// SIMATIC STEP 7 (V5.x) project Project
// CPU: CPU 315-2 DP
// CPU: CPU 315-2 DP
// station: Hardware
// station: SIMATIC 300(1)
// station: P_ADR_BUS
// station: Hardware
// station: SIMATIC 300(2)
// station: P_ADR_BUS
// station: _S7H_BUSSYSTEM_CT
// station: _S7H_BUSSYSTEM_CT
// program: S7 Program(1)
// program: S7 Program(1)

SYMBOL_TABLE
"A_Sensors"	DB 2	DB 2
"DI"	DB 3	DB 3
"SensorsSettings"	DB 4	DB 4
"Valves"	DB 5	DB 5
"BD_Coils"	DB 6	DB 6
"KB1_1_Coils"	DB 7	DB 7
"KB1_2_Coils"	DB 8	DB 8
"KB2_Coils"	DB 9	DB 9
"PO1_1_Coils"	DB 10	DB 10
"PO1_2_Coils"	DB 11	DB 11
"GA1_1_Coils"	DB 12	DB 12
"GA1_2_Coils"	DB 13	DB 13
"GA2_1_Coils"	DB 14	DB 14
"GA2_2_Coils"	DB 15	DB 15
"BD_AI_1"	DB 16	DB 16
"KB1_1_AI_1"	DB 17	DB 17
"KB1_1_AI_2"	DB 18	DB 18
"KB1_1_AI_3"	DB 19	DB 19
"KB1_2_AI_1"	DB 20	DB 20
"KB1_2_AI_2"	DB 21	DB 21
"KB1_2_AI_3"	DB 22	DB 22
"KB2_AI_1"	DB 23	DB 23
"KB2_AI_2"	DB 24	DB 24
"KB2_AI_3"	DB 25	DB 25
"KB2_AI_4"	DB 26	DB 26
"PO1_1_AI"	DB 27	DB 27
"PO1_2_AI"	DB 28	DB 28
"GA1_1_AI_1"	DB 29	DB 29
"GA1_1_AI_2"	DB 30	DB 30
"GA1_2_AI_1"	DB 31	DB 31
"GA1_2_AI_2"	DB 32	DB 32
"GA2_1_AI_1"	DB 33	DB 33
"GA2_1_AI_2"	DB 34	DB 34
"KD1_1_AI"	DB 35	DB 35
"GA2_2_AI_1"	DB 36	DB 36
"GA2_2_AI_2"	DB 37	DB 37
"KD1_1_AI_2"	DB 38	DB 38
"KD1_1_AI_3"	DB 39	DB 39
"KD1_1_AI_4"	DB 40	DB 40
"KD1_1_AI_5"	DB 41	DB 41
"KD1_1_Coils"	DB 42	DB 42
"BD1_ARR_AI"	DB 43	DB 43
"BD_AI_2"	DB 44	DB 44
"BD_AI_3"	DB 45	DB 45
"BD_DO_1"	DB 46	DB 46
"BD_DO_2"	DB 47	DB 47
"GA1_1_DO"	DB 48	DB 48
"GA1_2_DO"	DB 49	DB 49
"GA2_1_DO"	DB 50	DB 50
"GA2_2_DO"	DB 51	DB 51
"BD_REAL"	DB 52	DB 52
"KB1_1_REAL"	DB 53	DB 53
"KB1_2_REAL"	DB 54	DB 54
"KB2_REAL"	DB 55	DB 55
"PO1_1_REAL"	DB 56	DB 56
"PO1_2_REAL"	DB 57	DB 57
"GA1_1_REAL"	DB 58	DB 58
"GA1_2_REAL"	DB 59	DB 59
"GA2_1_REAL"	DB 60	DB 60
"GA2_2_REAL"	DB 61	DB 61
"KD_REAL"	DB 62	DB 62
"ModbusVars"	DB 63	DB 63
"BD_Outputs_1"	DB 64	DB 64
"BD_Outputs_2"	DB 65	DB 65
"PO1_1_Outputs"	DB 66	DB 66
"PO1_2_Outputs"	DB 67	DB 67
"GA1_1_Outputs"	DB 68	DB 68
"GA1_2_Outputs"	DB 69	DB 69
"GA2_1_Outputs"	DB 97	DB 97
"GA2_2_Outputs"	DB 98	DB 98
"BD_OutputBytes_1"	DB 99	DB 99
"BD_OutputBytes_2"	DB 111	DB 111
"PO1_1_OutBytes"	DB 112	DB 112
"PO1_2_OutBytes"	DB 113	DB 113
"GA1_1_OutBytes"	DB 114	DB 114
"GA1_2_OutBytes"	DB 115	DB 115
"GA2_1_OutBytes"	DB 116	DB 116
"GA2_2_OutBytes"	DB 117	DB 117
"StartStop"	DB 118	DB 118
"StartStopBytes"	DB 119	DB 119
"KB2_AI_Bearer"	DB 128	DB 128
"KB2_AI_Vibration"	DB 129	DB 129
"ModbusAddresses"	DB 130	DB 130
"PO2_AI"	DB 131	DB 131
"PO2_Reals"	DB 132	DB 132
"PO2_AI2"	DB 133	DB 133
"DI_Bytes"	DB 134	DB 134
"PCV10_PID_Vars"	DB 135	DB 135
"PCV21_PID_Vars"	DB 136	DB 136
"PCV22_PID_Vars"	DB 137	DB 137
"PCV25_PID_Vars"	DB 138	DB 138
"ValvesVars"	DB 139	DB 139
"SensorsAlarmSettings"	DB 140	DB 140
"BD_MaxMin"	DB 141	DB 141
"GA1_1_MinMax"	DB 142	DB 142
"GA1_2_MinMax"	DB 143	DB 143
"GA2_1_MinMax"	DB 144	DB 144
"GA2_2_MinMax"	DB 145	DB 145
"KB1_1_MinMax"	DB 146	DB 146
"KB1_2_MinMax"	DB 147	DB 147
"KD2_ManMax"	DB 148	DB 148
"PO1_1_MaxMin"	DB 149	DB 149
"PO1_2_MinMax"	DB 150	DB 150
"ProcessSettings"	DB 151	DB 151
"ProcessVars"	DB 152	DB 152
"PrepareStartStop"	DB 153	DB 153
"PO2_Coils"	DB 154	DB 154
"PO2_MinMax"	DB 155	DB 155
"SensorsErr"	DB 156	DB 156
"DB_DO"	DB 157	DB 157
"SensorsWarningSettings"	DB 158	DB 158
"VentVars"	DB 159	DB 159
"BD_Warnings"	DB 160	DB 160
"GA1_1_Warnings"	DB 161	DB 161
"GA1_2_Warnings"	DB 162	DB 162
"GA2_2_Warnings"	DB 163	DB 163
"GA2_1_Warnings"	DB 164	DB 164
"KB1_1_Warnings"	DB 165	DB 165
"KB1_2_Warnings"	DB 166	DB 166
"KD2_Warnings"	DB 167	DB 167
"KB2_MinMax"	DB 168	DB 168
"KB2_Warnings"	DB 169	DB 169
"PO1_1_Warnings"	DB 170	DB 170
"PO1_2_Warnings"	DB 171	DB 171
"PO2_Warnings"	DB 172	DB 172
"ModbusConnestions"	DB 173	DB 173
"KB2_Outputs"	DB 174	DB 174
"KB2_OutputBytes"	DB 175	DB 175
"KB2_CalcRealBytes"	DB 176	DB 176
"KB1_1_OutBytes"	DB 177	DB 177
"KB1_2_OutBytes"	DB 178	DB 178
"KB1_1_Outputs"	DB 179	DB 179
"KB1_2_Outputs"	DB 180	DB 180
"PO2_ArrCoils"	DB 181	DB 181
"KB2_ArrCoils"	DB 182	DB 182
"GA2_1_ArrCoils"	DB 183	DB 183
"GA2_2_ArrCoils"	DB 184	DB 184
"GA1_1_ArrCoils"	DB 185	DB 185
"GA1_2_ArrCoils"	DB 186	DB 186
"KB1_1_ArrCoils"	DB 187	DB 187
"KB1_2_ArrCoils"	DB 188	DB 188
"KD1_1_ArrCoils"	DB 189	DB 189
"PO1_1_ArrCoils"	DB 190	DB 190
"PO1_2_ArrCoils"	DB 191	DB 191
"BD_ArrCoils"	DB 192	DB 192
"AlmLocks"	DB 193	DB 193
"KB2_Resistance_Block"	DB 194	DB 194
"KB2_Resistance_Warn"	DB 195	DB 195
"GA2_2_AI_3"	DB 196	DB 196
"BlockVars"	DB 197	DB 197
"ValvesAutoManualStatus"	DB 198	DB 198
"GLV"	DB 301	DB 301
"ZB1"	DB 777	FB 38
"ZB2"	DB 778	FB 38
"ZB3"	DB 779	FB 38
"ZB4"	DB 780	FB 38
"ValvesPrgDB"	DB 781	FB 39
"KB2_AI_I_Motor"	DB 11120	DB 11120
"KB2_MotorMaxMin"	DB 11122	DB 11122
"KB2_MotorWarning"	DB 11123	DB 11123
"KB2_Motor"	DB 11199	DB 11199
"BD_GetReals"	FB 1	FB 1
"KB1_1_GetReals"	FB 2	FB 2
"KB1_2_GetReals"	FB 3	FB 3
"KB2_GetReals"	FB 4	FB 4
"PO1_1_GetReals"	FB 5	FB 5
"PO1_2_GetReals"	FB 6	FB 6
"P_RCV_RK"	FB 7	FB 7	// Receive Data / Provide Data
"P_SND_RK"	FB 8	FB 8	// Send Data / Fetch Data
"GA1_1_GetReal"	FB 9	FB 9
"MBMAREQ"	FB 10	FB 10	// MBMAREQ MODBUS MASTER REQUEST FUNCTION BLOCK
"GA1_2_GetReals"	FB 11	FB 11
"GA2_1_GetReals"	FB 12	FB 12
"GA2_2_GetReals"	FB 13	FB 13
"KD_GetReals"	FB 14	FB 14
"ModbusReal"	FB 15	FB 15
"ModbusCoils"	FB 16	FB 16
"ModbusOutputs"	FB 17	FB 17
"BD_GetOutputs"	FB 18	FB 18
"PO1_1_GetOutputs"	FB 19	FB 19
"PO1_2_GetOutputs"	FB 20	FB 20
"GA1_1_GetOutputs"	FB 21	FB 21
"GA1_2_GetOutputs"	FB 22	FB 22
"GA2_1_GetOutputs"	FB 23	FB 23
"GA2_2_GetOutputs"	FB 24	FB 24
"ModbusStartStop"	FB 25	FB 25
"GetStartStopBytes"	FB 26	FB 26
"GetAll"	FB 27	FB 27
"ModbusAll"	FB 28	FB 28
"InToVars"	FB 29	FB 29
"InToVarsST"	FB 30	FB 30
"PO2_GetReals"	FB 31	FB 31
"DI_ToVars"	FB 32	FB 32
"Valve_PID"	FB 33	FB 33
"fbPID"	FB 34	FB 34
"MBMA341"	FB 35	FB 35	// MBMA341 MODBUS MASTER COMMUNICATION FUNCTION BLOCK
"DERIVATIVE"	FB 36	FB 36
"INTEGRAL"	FB 37	FB 37
"DO_Valve"	FB 38	FB 38
"ValvesPrg"	FB 39	FB 39
"fbProcess_1"	FB 40	FB 40
"CONT_C"	FB 41	FB 41	// Continuous Control
"CONT_S"	FB 42	FB 42	// Step Control
"fbImpulsValve"	FB 43	FB 43
"fbImpulsValveSCL"	FB 44	FB 44
"prProcess"	FB 45	FB 45
"fbPO"	FB 46	FB 46
"fbKB"	FB 47	FB 47
"fbKZA"	FB 48	FB 48
"prDevices"	FB 49	FB 49
"GetCoils"	FB 50	FB 50
"Trash"	FB 51	FB 51
"VentBlock"	FB 52	FB 52
"KB2_GetOuts"	FB 53	FB 53
"fbStartStopProc"	FB 54	FB 54
"fbTON_New"	FB 55	FB 55
"fbStopDevices"	FB 56	FB 56
"fbN_O2_Block"	FB 57	FB 57
"TCONT_CP"	FB 58	FB 58	// temperature PID controller with pulse generator and self-tuning
"fbN_O2_Block_1"	FB 59	FB 59
"fbN_O2_Block_2"	FB 60	FB 60
"SET_SW_S"	FB 61	FB 61	// Set summer/winter time with status
"SWR_ZYK"	FB 101	FB 101	// Cyclic function block for Software Redundance
"SWR_SFCCOM"	FB 103	FB 103	// Communication function block for Software Redundance
"SWR_AG_COM"	FB 104	FB 104	// Communication function block for Software Redundance
"LinTrafo"	FC 1	FC 1
"fnWordPack"	FC 2	FC 2
"fnBytesToReal"	FC 3	FC 3
"fnBytesToRealOneComma"	FC 4	FC 4
"fnBytesToRealPressure"	FC 5	FC 5
"fnBytesToRealTwoComas"	FC 6	FC 6
"StartStopByte"	FC 7	FC 7
"LinTrafoInt"	FC 8	FC 8
"ByteToByte"	FC 9	FC 9
"fnRepeater"	FC 10	FC 10
"fnModbusCheckConnecrions"	FC 11	FC 11
"fnMicron"	FC 12	FC 12
"LinTrafoFlow"	FC 13	FC 13
"fnMaskByte"	FC 14	FC 14
"fnWordPackTwoComas"	FC 15	FC 15
"fnAverage"	FC 16	FC 16
"fnCbarPressure"	FC 17	FC 17
"SWR_START"	FC 100	FC 100	// Initialisation function for Software Redundance
"SWR_DIAG"	FC 102	FC 102	// Diagnostic function for Software Redundance
"_DI_XL1_QL3"	I 0.0	BOOL
"_DI_XL2_QL3"	I 0.1	BOOL
"_DI_Q3_Bad"	I 0.2	BOOL
"_DI_AB1_Working"	I 0.3	BOOL
"_DI_Kb_1_1_Working"	I 0.4	BOOL
"_DI_Kb_1_1_Alm"	I 0.5	BOOL
"_DI_Kb_1_2_Working"	I 0.6	BOOL
"_DI_Kb_1_2_Alm"	I 0.7	BOOL
"_DI_Kb_2_Working"	I 1.0	BOOL
"_DI_Kb_2_Alm"	I 1.1	BOOL
"_DI_Kd_1_Working"	I 1.2	BOOL
"_DI_Kd_1_Alm"	I 1.3	BOOL
"_DI_ZB_1_Opn"	I 1.4	BOOL
"_DI_ZB_1_Cls"	I 1.5	BOOL
"_DI_ZB_1_Local"	I 1.6	BOOL
"_DI_ZB_1_Alm"	I 1.7	BOOL
"_DI_ZB_2_Opn"	I 2.0	BOOL
"_DI_ZB_2_Cls"	I 2.1	BOOL
"_DI_ZB_2_Local"	I 2.2	BOOL
"_DI_ZB_2_Alm"	I 2.3	BOOL
"_DI_ZB_3_Opn"	I 2.4	BOOL
"_DI_ZB_3_Cls"	I 2.5	BOOL
"_DI_ZB_3_Local"	I 2.6	BOOL
"_DI_ZB_3_Alm"	I 2.7	BOOL
"_DI_EUV_001_Opn"	I 3.0	BOOL
"_DI_EUV_001_Cls"	I 3.1	BOOL
"_DI_EUV_001_Local"	I 3.2	BOOL
"_DI_EUV_001_Alm"	I 3.3	BOOL
"_DI_EUV_002_Opn"	I 3.4	BOOL
"_DI_EUV_002_Cls"	I 3.5	BOOL
"_DI_EUV_002_Local"	I 3.6	BOOL
"_DI_EUV_002_Alm"	I 3.7	BOOL
"_DI_EUV_003_Opn"	I 4.0	BOOL
"_DI_EUV_003_Cls"	I 4.1	BOOL
"_DI_EUV_003_Local"	I 4.2	BOOL
"_DI_EUV_003_Alm"	I 4.3	BOOL
"QSA_19_1_1"	I 4.4	BOOL
"QSA_23_1_1"	I 4.5	BOOL
"QSA_19_1_2"	I 4.6	BOOL
"QSA_23_1_2"	I 4.7	BOOL
"QSA_19_1_3"	I 5.0	BOOL
"QSA_23_1_3"	I 5.1	BOOL
"QSA_19_1_4"	I 5.2	BOOL
"QSA_23_1_4"	I 5.3	BOOL
"QSA_19_1_5"	I 5.4	BOOL
"QSA_23_1_5"	I 5.5	BOOL
"Q3_BAD"	I 5.6	BOOL
"AB_1_Alm"	I 5.7	BOOL
"AB_2_Working"	I 6.0	BOOL
"AB_2_Alm"	I 6.1	BOOL
"AB_3_Working"	I 6.2	BOOL
"AB_3_Alm"	I 6.3	BOOL
"AB_4_Working"	I 6.4	BOOL
"AB_4_Alm"	I 6.5	BOOL
"P2_Alm"	I 6.6	BOOL
"P2_Working"	I 6.7	BOOL
"P3_Alm"	I 7.0	BOOL
"P3_Working"	I 7.1	BOOL
"IBP_1_Working"	I 7.2	BOOL
"IBP_1_Alm"	I 7.3	BOOL
"IBP_1_Bypas"	I 7.4	BOOL
"IBP_2_Working"	I 7.5	BOOL
"IBP_2_Alm"	I 7.6	BOOL
"IBP_2_Bypas"	I 7.7	BOOL
"_DI_ZB_4_Opn"	I 8.0	BOOL
"_DI_ZB_4_Cls"	I 8.1	BOOL
"_DI_ZB_4_Local"	I 8.2	BOOL
"_DI_ZB_4_Alm"	I 8.3	BOOL
"XL1_Q4"	I 8.4	BOOL
"XL2_Q4"	I 8.5	BOOL
"Q4_BAD"	I 8.6	BOOL
"_KB_1_1_1PIR7"	IW 256	WORD
"_KB_1_2_2PIR7"	IW 258	WORD
"_1PIR6"	IW 260	WORD
"_KZA_1_2_2PIR6"	IW 262	WORD
"_KB_2_PIR8"	IW 264	WORD
"_1PIR20"	IW 266	WORD
"_2PIR20"	IW 268	WORD
"_TIR10"	IW 270	WORD
"_FIR10"	IW 272	WORD
"_PIR5"	IW 274	WORD
"_FIR5"	IW 276	WORD
"_PIRC21"	IW 278	WORD
"_1PIR27"	IW 280	WORD
"_QIRAH3"	IW 282	WORD
"_2PIR27"	IW 284	WORD
"_PIR4"	IW 286	WORD
"_FIR_4"	IW 288	WORD
"_PIRC22"	IW 290	WORD
"_PIRC23"	IW 292	WORD
"_PIRC24"	IW 294	WORD
"_PIRC25"	IW 296	WORD
"_FIR_25"	IW 298	WORD
"_1PIRC26"	IW 300	WORD
"_2PIRC26"	IW 302	WORD
"_C10"	IW 304	WORD
"_TIR5"	IW 306	WORD
"_TIR4"	IW 308	WORD
"_TIR25"	IW 310	WORD
"_AIR1"	IW 312	WORD
"_QIRAH4Q4"	IW 314	WORD
"CYC_INT5"	OB 35	OB 35	// Cyclic Interrupt 5
"CYCL_FLT"	OB 80	OB 80	// Cycle Time Fault
"I/O_FLT1"	OB 82	OB 82	// I/O Point Fault 1
"OBNL_FLT"	OB 85	OB 85	// OB Not Loaded Fault
"RACK_FLT"	OB 86	OB 86	// Loss of Rack Fault
"COMM_FLT"	OB 87	OB 87	// Communication Fault
"COMPLETE RESTART"	OB 100	OB 100	// Complete Restart
"PROG_ERR"	OB 121	OB 121	// Programming Error
"MOD_ERR"	OB 122	OB 122	// Module Access Error
"_DO_HS1Q1_Acknow"	Q 0.0	BOOL
"_DO_HS1Q1_Check"	Q 0.1	BOOL
"_DO_KB_1_1_Stop"	Q 0.2	BOOL
"_DO_KB_1_1_Start"	Q 0.3	BOOL
"_DO_KB_1_2_Stop"	Q 0.4	BOOL
"_DO_KB_1_2_Start"	Q 0.5	BOOL
"_DO_KB_2_Stop"	Q 0.6	BOOL
"_DO_KB_2_Start"	Q 0.7	BOOL
"_DO_KD_1_Start"	Q 1.0	BOOL
"_DO_KD_1_Stop"	Q 1.1	BOOL
"_DO_ZB_1_CmdOpn"	Q 1.2	BOOL
"_DO_ZB_1_CmdCls"	Q 1.3	BOOL
"_DO_ZB_1_CmdStop"	Q 1.4	BOOL
"_DO_ZB_2_CmdOpn"	Q 1.5	BOOL
"_DO_ZB_2_CmdCls"	Q 1.6	BOOL
"_DO_ZB_2_CmdStop"	Q 1.7	BOOL
"_DO_ZB_3_CmdOpn"	Q 2.0	BOOL
"_DO_ZB_3_CmdCls"	Q 2.1	BOOL
"_DO_ZB_3_CmdStop"	Q 2.2	BOOL
"_DO_AlnVent"	Q 2.3	BOOL
"_DO_ZB_4_CmdOpn"	Q 2.4	BOOL
"_DO_ZB_4_CmdCls"	Q 2.5	BOOL
"_DO_ZB_4_CmdStop"	Q 2.6	BOOL
"_AO_N_Set_PCV10"	QW 256	WORD
"_AO_N_Set_PCV21"	QW 258	WORD
"_AO_Air_Set_PCV22"	QW 260	WORD
"_AO_Air_Set_PCV25"	QW 262	WORD
"TP"	SFB 3	SFB 3	// Generate a Pulse
"RDREC"	SFB 52	SFB 52	// Read a Process Data Record
"WRREC"	SFB 53	SFB 53	// Write a Process Data Record
"READ_CLK"	SFC 1	SFC 1	// Read System Clock
"GADR_LGC"	SFC 5	SFC 5	// Query Logical Address of a Channel
"RD_SINFO"	SFC 6	SFC 6	// Read OB Start Information
"DP_PRAL"	SFC 7	SFC 7	// Triggering a Hardware Interrupt on the DP Master
"EN_MSG"	SFC 9	SFC 9	// Enable Block-Related, Symbol-Related and Group Status Messages
"DIS_MSG"	SFC 10	SFC 10	// Disable Block-Related, Symbol-Related and Group Status Messages
"DPSYC_FR"	SFC 11	SFC 11	// Sending Control Commands to Groups of DP Slaves
"DPNRM_DG"	SFC 13	SFC 13	// Read Diagnostic Data of a DP Slave
"DPRD_DAT"	SFC 14	SFC 14	// Read Consistent Data of a Standard DP Slave
"DPWR_DAT"	SFC 15	SFC 15	// Write Consistent Data to a Standard DP Slave
"ALARM_SQ"	SFC 17	SFC 17	// Generate Block-Related Messages with Acknowledgment
"ALARM_S"	SFC 18	SFC 18	// Generate Permanently Acknowledged Block-Related Messages
"ALARM_SC"	SFC 19	SFC 19	// Query the Acknowledgment Status of the last ALARM_SQ Entering State Message
"BLKMOV"	SFC 20	SFC 20	// Copy Variables
"FILL"	SFC 21	SFC 21	// Initialize a Memory Area
"CREAT_DB"	SFC 22	SFC 22	// Create Data Block
"DEL_DB"	SFC 23	SFC 23	// Delete Data Block
"TEST_DB"	SFC 24	SFC 24	// Test Data Block
"COMPRESS"	SFC 25	SFC 25	// Compress the User Memory
"UPDAT_PI"	SFC 26	SFC 26	// Update Process Image Input
"UPDAT_PO"	SFC 27	SFC 27	// Update Outputs on I/O Module
"SET_TINT"	SFC 28	SFC 28	// Set Time-of-Day Interrupt
"CAN_TINT"	SFC 29	SFC 29	// Cancel Time-of-Day Interrupt
"ACT_TINT"	SFC 30	SFC 30	// Activate Time-of-Day Interrupt
"QRY_TINT"	SFC 31	SFC 31	// Query Time-of-Day Interrupt
"SRT_DINT"	SFC 32	SFC 32	// Start Time-Delay Interrupt
"CAN_DINT"	SFC 33	SFC 33	// Cancel Time-Delay Interrupt
"QRY_DINT"	SFC 34	SFC 34	// Query Time-Delay Interrupt
"MP_ALM"	SFC 35	SFC 35	// Trigger Multicomputing Interrupt
"MSK_FLT"	SFC 36	SFC 36	// Mask Synchronous Errors
"DMSK_FLT"	SFC 37	SFC 37	// Unmask Synchronous Errors
"READ_ERR"	SFC 38	SFC 38	// Read Error Registers
"DIS_IRT"	SFC 39	SFC 39	// Disable New Interrupts and Asynchronous Errors
"EN_IRT"	SFC 40	SFC 40	// Enable New Interrupts and Asynchronous Errors
"DIS_AIRT"	SFC 41	SFC 41	// Delay the Higher Priority Interrupts and Asynchronous Errors
"EN_AIRT"	SFC 42	SFC 42	// Enable Higher Priority Interrupts and Asynchronous Errors
"RE_TRIGR"	SFC 43	SFC 43	// Retrigger Cycle Time Monitoring
"REPL_VAL"	SFC 44	SFC 44	// Transfer Substitute Value to Accumulator 1
"STP"	SFC 46	SFC 46	// Change the CPU to STOP
"WAIT"	SFC 47	SFC 47	// Delay Execution of the User Program
"SNC_RTCB"	SFC 48	SFC 48	// Synchronize Slave Clocks
"LGC_GADR"	SFC 49	SFC 49	// Query the Module Slot Belonging to a Logical Address
"RD_LGADR"	SFC 50	SFC 50	// Read All Logical Addresses of a Module
"RDSYSST"	SFC 51	SFC 51	// Read a System Status List or Partial List
"WR_USMSG"	SFC 52	SFC 52	// Write a User-Defined Diagnostic Event to the Diagnostic Buffer
"RD_DPARM"	SFC 54	SFC 54	// Reading Predefined Parameters
"WR_PARM"	SFC 55	SFC 55	// Write Dynamic Parameters
"WR_DPARM"	SFC 56	SFC 56	// Write Default Parameters
"PARM_MOD"	SFC 57	SFC 57	// Assign Parameters to a Module
"WR_REC"	SFC 58	SFC 58	// Write Data Record
"RD_REC"	SFC 59	SFC 59	// Read a Data Record
"GD_SND"	SFC 60	SFC 60	// Send a GD Packet
"GD_RCV"	SFC 61	SFC 61	// Fetch a Received GD Packet
"CONTROL"	SFC 62	SFC 62	// Query the Status of a Connection Belonging to a Communication SFB Instance
"AB_CALL"	SFC 63	SFC 63	// Assembly Code Block (CPU 614)
"TIME_TCK"	SFC 64	SFC 64	// Read the System Time
"X_SEND"	SFC 65	SFC 65	// Send Data to a Communication Partner outside the Local S7 Station
"X_RCV"	SFC 66	SFC 66	// Receive Data from a Communication Partner outside the Local S7 Station
"X_GET"	SFC 67	SFC 67	// Read Data from a Communication Partner outside the Local S7 Station
"X_PUT"	SFC 68	SFC 68	// Write Data to a Communication Partner outside the Local S7 Station
"X_ABORT"	SFC 69	SFC 69	// Abort an Existing Connection to a  Partner outside the Local S7 Station
"I_GET"	SFC 72	SFC 72	// Read Data from a Communication Partner within the Local S7 Station
"I_PUT"	SFC 73	SFC 73	// Write Data to a Communication Partner within the Local S7 Station
"I_ABORT"	SFC 74	SFC 74	// Abort an Existing Connection to a Partner within the Local S7 Station
"DI_Vars"	VAT 1	
"DO_Vars"	VAT 2	
"AI_Vars"	VAT 3	
"AO_Vars"	VAT 4	
END_SYMBOL_TABLE

SYMBOL_TABLE
"A_Sensors"	DB 2	DB 2
"DI"	DB 3	DB 3
"SensorsSettings"	DB 4	DB 4
"Valves"	DB 5	DB 5
"BD_Coils"	DB 6	DB 6
"KB1_1_Coils"	DB 7	DB 7
"KB1_2_Coils"	DB 8	DB 8
"KB2_Coils"	DB 9	DB 9
"PO1_1_Coils"	DB 10	DB 10
"PO1_2_Coils"	DB 11	DB 11
"GA1_1_Coils"	DB 12	DB 12
"GA1_2_Coils"	DB 13	DB 13
"GA2_1_Coils"	DB 14	DB 14
"GA2_2_Coils"	DB 15	DB 15
"BD_AI_1"	DB 16	DB 16
"KB1_1_AI_1"	DB 17	DB 17
"KB1_1_AI_2"	DB 18	DB 18
"KB1_1_AI_3"	DB 19	DB 19
"KB1_2_AI_1"	DB 20	DB 20
"KB1_2_AI_2"	DB 21	DB 21
"KB1_2_AI_3"	DB 22	DB 22
"KB2_AI_1"	DB 23	DB 23
"KB2_AI_2"	DB 24	DB 24
"KB2_AI_3"	DB 25	DB 25
"KB2_AI_4"	DB 26	DB 26
"PO1_1_AI"	DB 27	DB 27
"PO1_2_AI"	DB 28	DB 28
"GA1_1_AI_1"	DB 29	DB 29
"GA1_1_AI_2"	DB 30	DB 30
"GA1_2_AI_1"	DB 31	DB 31
"GA1_2_AI_2"	DB 32	DB 32
"GA2_1_AI_1"	DB 33	DB 33
"GA2_1_AI_2"	DB 34	DB 34
"KD1_1_AI"	DB 35	DB 35
"GA2_2_AI_1"	DB 36	DB 36
"GA2_2_AI_2"	DB 37	DB 37
"KD1_1_AI_2"	DB 38	DB 38
"KD1_1_AI_3"	DB 39	DB 39
"KD1_1_AI_4"	DB 40	DB 40
"KD1_1_AI_5"	DB 41	DB 41
"KD1_1_Coils"	DB 42	DB 42
"BD1_ARR_AI"	DB 43	DB 43
"BD_AI_2"	DB 44	DB 44
"BD_AI_3"	DB 45	DB 45
"BD_DO_1"	DB 46	DB 46
"BD_DO_2"	DB 47	DB 47
"GA1_1_DO"	DB 48	DB 48
"GA1_2_DO"	DB 49	DB 49
"GA2_1_DO"	DB 50	DB 50
"GA2_2_DO"	DB 51	DB 51
"BD_REAL"	DB 52	DB 52
"KB1_1_REAL"	DB 53	DB 53
"KB1_2_REAL"	DB 54	DB 54
"KB2_REAL"	DB 55	DB 55
"PO1_1_REAL"	DB 56	DB 56
"PO1_2_REAL"	DB 57	DB 57
"GA1_1_REAL"	DB 58	DB 58
"GA1_2_REAL"	DB 59	DB 59
"GA2_1_REAL"	DB 60	DB 60
"GA2_2_REAL"	DB 61	DB 61
"KD_REAL"	DB 62	DB 62
"ModbusVars"	DB 63	DB 63
"BD_Outputs_1"	DB 64	DB 64
"BD_Outputs_2"	DB 65	DB 65
"PO1_1_Outputs"	DB 66	DB 66
"PO1_2_Outputs"	DB 67	DB 67
"GA1_1_Outputs"	DB 68	DB 68
"GA1_2_Outputs"	DB 69	DB 69
"GA2_1_Outputs"	DB 97	DB 97
"GA2_2_Outputs"	DB 98	DB 98
"BD_OutputBytes_1"	DB 99	DB 99
"BD_OutputBytes_2"	DB 111	DB 111
"PO1_1_OutBytes"	DB 112	DB 112
"PO1_2_OutBytes"	DB 113	DB 113
"GA1_1_OutBytes"	DB 114	DB 114
"GA1_2_OutBytes"	DB 115	DB 115
"GA2_1_OutBytes"	DB 116	DB 116
"GA2_2_OutBytes"	DB 117	DB 117
"StartStop"	DB 118	DB 118
"StartStopBytes"	DB 119	DB 119
"KB2_AI_Bearer"	DB 128	DB 128
"KB2_AI_Vibration"	DB 129	DB 129
"ModbusAddresses"	DB 130	DB 130
"PO2_AI"	DB 131	DB 131
"PO2_Reals"	DB 132	DB 132
"PO2_AI2"	DB 133	DB 133
"DI_Bytes"	DB 134	DB 134
"PCV10_PID_Vars"	DB 135	DB 135
"PCV21_PID_Vars"	DB 136	DB 136
"PCV22_PID_Vars"	DB 137	DB 137
"PCV25_PID_Vars"	DB 138	DB 138
"ValvesVars"	DB 139	DB 139
"SensorsAlarmSettings"	DB 140	DB 140
"BD_MaxMin"	DB 141	DB 141
"GA1_1_MinMax"	DB 142	DB 142
"GA1_2_MinMax"	DB 143	DB 143
"GA2_1_MinMax"	DB 144	DB 144
"GA2_2_MinMax"	DB 145	DB 145
"KB1_1_MinMax"	DB 146	DB 146
"KB1_2_MinMax"	DB 147	DB 147
"KD2_ManMax"	DB 148	DB 148
"PO1_1_MaxMin"	DB 149	DB 149
"PO1_2_MinMax"	DB 150	DB 150
"ProcessSettings"	DB 151	DB 151
"ProcessVars"	DB 152	DB 152
"PrepareStartStop"	DB 153	DB 153
"PO2_Coils"	DB 154	DB 154
"PO2_MinMax"	DB 155	DB 155
"SensorsErr"	DB 156	DB 156
"DB_DO"	DB 157	DB 157
"SensorsWarningSettings"	DB 158	DB 158
"VentVars"	DB 159	DB 159
"BD_Warnings"	DB 160	DB 160
"GA1_1_Warnings"	DB 161	DB 161
"GA1_2_Warnings"	DB 162	DB 162
"GA2_2_Warnings"	DB 163	DB 163
"GA2_1_Warnings"	DB 164	DB 164
"KB1_1_Warnings"	DB 165	DB 165
"KB1_2_Warnings"	DB 166	DB 166
"KD2_Warnings"	DB 167	DB 167
"KB2_MinMax"	DB 168	DB 168
"KB2_Warnings"	DB 169	DB 169
"PO1_1_Warnings"	DB 170	DB 170
"PO1_2_Warnings"	DB 171	DB 171
"PO2_Warnings"	DB 172	DB 172
"ModbusConnestions"	DB 173	DB 173
"KB2_Outputs"	DB 174	DB 174
"KB2_OutputBytes"	DB 175	DB 175
"KB2_CalcRealBytes"	DB 176	DB 176
"KB1_1_OutBytes"	DB 177	DB 177
"KB1_2_OutBytes"	DB 178	DB 178
"KB1_1_Outputs"	DB 179	DB 179
"KB1_2_Outputs"	DB 180	DB 180
"PO2_ArrCoils"	DB 181	DB 181
"KB2_ArrCoils"	DB 182	DB 182
"GA2_1_ArrCoils"	DB 183	DB 183
"GA2_2_ArrCoils"	DB 184	DB 184
"GA1_1_ArrCoils"	DB 185	DB 185
"GA1_2_ArrCoils"	DB 186	DB 186
"KB1_1_ArrCoils"	DB 187	DB 187
"KB1_2_ArrCoils"	DB 188	DB 188
"KD1_1_ArrCoils"	DB 189	DB 189
"PO1_1_ArrCoils"	DB 190	DB 190
"PO1_2_ArrCoils"	DB 191	DB 191
"BD_ArrCoils"	DB 192	DB 192
"AlmLocks"	DB 193	DB 193
"KB2_Resistance_Block"	DB 194	DB 194
"KB2_Resistance_Warn"	DB 195	DB 195
"GA2_2_AI_3"	DB 196	DB 196
"BlockVars"	DB 197	DB 197
"ValvesAutoManualStatus"	DB 198	DB 198
"GLV"	DB 301	DB 301
"ZB1"	DB 777	FB 38
"ZB2"	DB 778	FB 38
"ZB3"	DB 779	FB 38
"ZB4"	DB 780	FB 38
"ValvesPrgDB"	DB 781	FB 39
"KB2_AI_I_Motor"	DB 11120	DB 11120
"KB2_MotorMaxMin"	DB 11122	DB 11122
"KB2_MotorWarning"	DB 11123	DB 11123
"KB2_Motor"	DB 11199	DB 11199
"BD_GetReals"	FB 1	FB 1
"KB1_1_GetReals"	FB 2	FB 2
"KB1_2_GetReals"	FB 3	FB 3
"KB2_GetReals"	FB 4	FB 4
"PO1_1_GetReals"	FB 5	FB 5
"PO1_2_GetReals"	FB 6	FB 6
"P_RCV_RK"	FB 7	FB 7	// Receive Data / Provide Data
"P_SND_RK"	FB 8	FB 8	// Send Data / Fetch Data
"GA1_1_GetReal"	FB 9	FB 9
"MBMAREQ"	FB 10	FB 10	// MBMAREQ MODBUS MASTER REQUEST FUNCTION BLOCK
"GA1_2_GetReals"	FB 11	FB 11
"GA2_1_GetReals"	FB 12	FB 12
"GA2_2_GetReals"	FB 13	FB 13
"KD_GetReals"	FB 14	FB 14
"ModbusReal"	FB 15	FB 15
"ModbusCoils"	FB 16	FB 16
"ModbusOutputs"	FB 17	FB 17
"BD_GetOutputs"	FB 18	FB 18
"PO1_1_GetOutputs"	FB 19	FB 19
"PO1_2_GetOutputs"	FB 20	FB 20
"GA1_1_GetOutputs"	FB 21	FB 21
"GA1_2_GetOutputs"	FB 22	FB 22
"GA2_1_GetOutputs"	FB 23	FB 23
"GA2_2_GetOutputs"	FB 24	FB 24
"ModbusStartStop"	FB 25	FB 25
"GetStartStopBytes"	FB 26	FB 26
"GetAll"	FB 27	FB 27
"ModbusAll"	FB 28	FB 28
"InToVars"	FB 29	FB 29
"InToVarsST"	FB 30	FB 30
"PO2_GetReals"	FB 31	FB 31
"DI_ToVars"	FB 32	FB 32
"Valve_PID"	FB 33	FB 33
"fbPID"	FB 34	FB 34
"MBMA341"	FB 35	FB 35	// MBMA341 MODBUS MASTER COMMUNICATION FUNCTION BLOCK
"DERIVATIVE"	FB 36	FB 36
"INTEGRAL"	FB 37	FB 37
"DO_Valve"	FB 38	FB 38
"ValvesPrg"	FB 39	FB 39
"fbProcess_1"	FB 40	FB 40
"CONT_C"	FB 41	FB 41	// Continuous Control
"CONT_S"	FB 42	FB 42	// Step Control
"fbImpulsValve"	FB 43	FB 43
"fbImpulsValveSCL"	FB 44	FB 44
"prProcess"	FB 45	FB 45
"fbPO"	FB 46	FB 46
"fbKB"	FB 47	FB 47
"fbKZA"	FB 48	FB 48
"prDevices"	FB 49	FB 49
"GetCoils"	FB 50	FB 50
"Trash"	FB 51	FB 51
"VentBlock"	FB 52	FB 52
"KB2_GetOuts"	FB 53	FB 53
"fbStartStopProc"	FB 54	FB 54
"fbTON_New"	FB 55	FB 55
"fbStopDevices"	FB 56	FB 56
"fbN_O2_Block"	FB 57	FB 57
"TCONT_CP"	FB 58	FB 58	// temperature PID controller with pulse generator and self-tuning
"fbN_O2_Block_1"	FB 59	FB 59
"fbN_O2_Block_2"	FB 60	FB 60
"SET_SW_S"	FB 61	FB 61	// Set summer/winter time with status
"SWR_ZYK"	FB 101	FB 101	// Cyclic function block for Software Redundance
"SWR_SFCCOM"	FB 103	FB 103	// Communication function block for Software Redundance
"SWR_AG_COM"	FB 104	FB 104	// Communication function block for Software Redundance
"LinTrafo"	FC 1	FC 1
"fnWordPack"	FC 2	FC 2
"fnBytesToReal"	FC 3	FC 3
"fnBytesToRealOneComma"	FC 4	FC 4
"fnBytesToRealPressure"	FC 5	FC 5
"fnBytesToRealTwoComas"	FC 6	FC 6
"StartStopByte"	FC 7	FC 7
"LinTrafoInt"	FC 8	FC 8
"ByteToByte"	FC 9	FC 9
"fnRepeater"	FC 10	FC 10
"fnModbusCheckConnecrions"	FC 11	FC 11
"fnMicron"	FC 12	FC 12
"LinTrafoFlow"	FC 13	FC 13
"fnMaskByte"	FC 14	FC 14
"fnWordPackTwoComas"	FC 15	FC 15
"fnAverage"	FC 16	FC 16
"fnCbarPressure"	FC 17	FC 17
"SWR_START"	FC 100	FC 100	// Initialisation function for Software Redundance
"SWR_DIAG"	FC 102	FC 102	// Diagnostic function for Software Redundance
"_DI_XL1_QL3"	I 0.0	BOOL
"_DI_XL2_QL3"	I 0.1	BOOL
"_DI_Q3_Bad"	I 0.2	BOOL
"_DI_AB1_Working"	I 0.3	BOOL
"_DI_Kb_1_1_Working"	I 0.4	BOOL
"_DI_Kb_1_1_Alm"	I 0.5	BOOL
"_DI_Kb_1_2_Working"	I 0.6	BOOL
"_DI_Kb_1_2_Alm"	I 0.7	BOOL
"_DI_Kb_2_Working"	I 1.0	BOOL
"_DI_Kb_2_Alm"	I 1.1	BOOL
"_DI_Kd_1_Working"	I 1.2	BOOL
"_DI_Kd_1_Alm"	I 1.3	BOOL
"_DI_ZB_1_Opn"	I 1.4	BOOL
"_DI_ZB_1_Cls"	I 1.5	BOOL
"_DI_ZB_1_Local"	I 1.6	BOOL
"_DI_ZB_1_Alm"	I 1.7	BOOL
"_DI_ZB_2_Opn"	I 2.0	BOOL
"_DI_ZB_2_Cls"	I 2.1	BOOL
"_DI_ZB_2_Local"	I 2.2	BOOL
"_DI_ZB_2_Alm"	I 2.3	BOOL
"_DI_ZB_3_Opn"	I 2.4	BOOL
"_DI_ZB_3_Cls"	I 2.5	BOOL
"_DI_ZB_3_Local"	I 2.6	BOOL
"_DI_ZB_3_Alm"	I 2.7	BOOL
"_DI_EUV_001_Opn"	I 3.0	BOOL
"_DI_EUV_001_Cls"	I 3.1	BOOL
"_DI_EUV_001_Local"	I 3.2	BOOL
"_DI_EUV_001_Alm"	I 3.3	BOOL
"_DI_EUV_002_Opn"	I 3.4	BOOL
"_DI_EUV_002_Cls"	I 3.5	BOOL
"_DI_EUV_002_Local"	I 3.6	BOOL
"_DI_EUV_002_Alm"	I 3.7	BOOL
"_DI_EUV_003_Opn"	I 4.0	BOOL
"_DI_EUV_003_Cls"	I 4.1	BOOL
"_DI_EUV_003_Local"	I 4.2	BOOL
"_DI_EUV_003_Alm"	I 4.3	BOOL
"QSA_19_1_1"	I 4.4	BOOL
"QSA_23_1_1"	I 4.5	BOOL
"QSA_19_1_2"	I 4.6	BOOL
"QSA_23_1_2"	I 4.7	BOOL
"QSA_19_1_3"	I 5.0	BOOL
"QSA_23_1_3"	I 5.1	BOOL
"QSA_19_1_4"	I 5.2	BOOL
"QSA_23_1_4"	I 5.3	BOOL
"QSA_19_1_5"	I 5.4	BOOL
"QSA_23_1_5"	I 5.5	BOOL
"Q3_BAD"	I 5.6	BOOL
"AB_1_Alm"	I 5.7	BOOL
"AB_2_Working"	I 6.0	BOOL
"AB_2_Alm"	I 6.1	BOOL
"AB_3_Working"	I 6.2	BOOL
"AB_3_Alm"	I 6.3	BOOL
"AB_4_Working"	I 6.4	BOOL
"AB_4_Alm"	I 6.5	BOOL
"P2_Alm"	I 6.6	BOOL
"P2_Working"	I 6.7	BOOL
"P3_Alm"	I 7.0	BOOL
"P3_Working"	I 7.1	BOOL
"IBP_1_Working"	I 7.2	BOOL
"IBP_1_Alm"	I 7.3	BOOL
"IBP_1_Bypas"	I 7.4	BOOL
"IBP_2_Working"	I 7.5	BOOL
"IBP_2_Alm"	I 7.6	BOOL
"IBP_2_Bypas"	I 7.7	BOOL
"_DI_ZB_4_Opn"	I 8.0	BOOL
"_DI_ZB_4_Cls"	I 8.1	BOOL
"_DI_ZB_4_Local"	I 8.2	BOOL
"_DI_ZB_4_Alm"	I 8.3	BOOL
"XL1_Q4"	I 8.4	BOOL
"XL2_Q4"	I 8.5	BOOL
"Q4_BAD"	I 8.6	BOOL
"_KB_1_1_1PIR7"	IW 256	WORD
"_KB_1_2_2PIR7"	IW 258	WORD
"_1PIR6"	IW 260	WORD
"_KZA_1_2_2PIR6"	IW 262	WORD
"_KB_2_PIR8"	IW 264	WORD
"_1PIR20"	IW 266	WORD
"_2PIR20"	IW 268	WORD
"_TIR10"	IW 270	WORD
"_FIR10"	IW 272	WORD
"_PIR5"	IW 274	WORD
"_FIR5"	IW 276	WORD
"_PIRC21"	IW 278	WORD
"_1PIR27"	IW 280	WORD
"_QIRAH3"	IW 282	WORD
"_2PIR27"	IW 284	WORD
"_PIR4"	IW 286	WORD
"_FIR_4"	IW 288	WORD
"_PIRC22"	IW 290	WORD
"_PIRC23"	IW 292	WORD
"_PIRC24"	IW 294	WORD
"_PIRC25"	IW 296	WORD
"_FIR_25"	IW 298	WORD
"_1PIRC26"	IW 300	WORD
"_2PIRC26"	IW 302	WORD
"_C10"	IW 304	WORD
"_TIR5"	IW 306	WORD
"_TIR4"	IW 308	WORD
"_TIR25"	IW 310	WORD
"_AIR1"	IW 312	WORD
"_QIRAH4Q4"	IW 314	WORD
"CYC_INT5"	OB 35	OB 35	// Cyclic Interrupt 5
"CYCL_FLT"	OB 80	OB 80	// Cycle Time Fault
"I/O_FLT1"	OB 82	OB 82	// I/O Point Fault 1
"OBNL_FLT"	OB 85	OB 85	// OB Not Loaded Fault
"RACK_FLT"	OB 86	OB 86	// Loss of Rack Fault
"COMM_FLT"	OB 87	OB 87	// Communication Fault
"COMPLETE RESTART"	OB 100	OB 100	// Complete Restart
"PROG_ERR"	OB 121	OB 121	// Programming Error
"MOD_ERR"	OB 122	OB 122	// Module Access Error
"_DO_HS1Q1_Acknow"	Q 0.0	BOOL
"_DO_HS1Q1_Check"	Q 0.1	BOOL
"_DO_KB_1_1_Stop"	Q 0.2	BOOL
"_DO_KB_1_1_Start"	Q 0.3	BOOL
"_DO_KB_1_2_Stop"	Q 0.4	BOOL
"_DO_KB_1_2_Start"	Q 0.5	BOOL
"_DO_KB_2_Stop"	Q 0.6	BOOL
"_DO_KB_2_Start"	Q 0.7	BOOL
"_DO_KD_1_Start"	Q 1.0	BOOL
"_DO_KD_1_Stop"	Q 1.1	BOOL
"_DO_ZB_1_CmdOpn"	Q 1.2	BOOL
"_DO_ZB_1_CmdCls"	Q 1.3	BOOL
"_DO_ZB_1_CmdStop"	Q 1.4	BOOL
"_DO_ZB_2_CmdOpn"	Q 1.5	BOOL
"_DO_ZB_2_CmdCls"	Q 1.6	BOOL
"_DO_ZB_2_CmdStop"	Q 1.7	BOOL
"_DO_ZB_3_CmdOpn"	Q 2.0	BOOL
"_DO_ZB_3_CmdCls"	Q 2.1	BOOL
"_DO_ZB_3_CmdStop"	Q 2.2	BOOL
"_DO_AlnVent"	Q 2.3	BOOL
"_DO_ZB_4_CmdOpn"	Q 2.4	BOOL
"_DO_ZB_4_CmdCls"	Q 2.5	BOOL
"_DO_ZB_4_CmdStop"	Q 2.6	BOOL
"_AO_N_Set_PCV10"	QW 256	WORD
"_AO_N_Set_PCV21"	QW 258	WORD
"_AO_Air_Set_PCV22"	QW 260	WORD
"_AO_Air_Set_PCV25"	QW 262	WORD
"TP"	SFB 3	SFB 3	// Generate a Pulse
"RDREC"	SFB 52	SFB 52	// Read a Process Data Record
"WRREC"	SFB 53	SFB 53	// Write a Process Data Record
"READ_CLK"	SFC 1	SFC 1	// Read System Clock
"GADR_LGC"	SFC 5	SFC 5	// Query Logical Address of a Channel
"RD_SINFO"	SFC 6	SFC 6	// Read OB Start Information
"DP_PRAL"	SFC 7	SFC 7	// Triggering a Hardware Interrupt on the DP Master
"EN_MSG"	SFC 9	SFC 9	// Enable Block-Related, Symbol-Related and Group Status Messages
"DIS_MSG"	SFC 10	SFC 10	// Disable Block-Related, Symbol-Related and Group Status Messages
"DPSYC_FR"	SFC 11	SFC 11	// Sending Control Commands to Groups of DP Slaves
"DPNRM_DG"	SFC 13	SFC 13	// Read Diagnostic Data of a DP Slave
"DPRD_DAT"	SFC 14	SFC 14	// Read Consistent Data of a Standard DP Slave
"DPWR_DAT"	SFC 15	SFC 15	// Write Consistent Data to a Standard DP Slave
"ALARM_SQ"	SFC 17	SFC 17	// Generate Block-Related Messages with Acknowledgment
"ALARM_S"	SFC 18	SFC 18	// Generate Permanently Acknowledged Block-Related Messages
"ALARM_SC"	SFC 19	SFC 19	// Query the Acknowledgment Status of the last ALARM_SQ Entering State Message
"BLKMOV"	SFC 20	SFC 20	// Copy Variables
"FILL"	SFC 21	SFC 21	// Initialize a Memory Area
"CREAT_DB"	SFC 22	SFC 22	// Create Data Block
"DEL_DB"	SFC 23	SFC 23	// Delete Data Block
"TEST_DB"	SFC 24	SFC 24	// Test Data Block
"COMPRESS"	SFC 25	SFC 25	// Compress the User Memory
"UPDAT_PI"	SFC 26	SFC 26	// Update Process Image Input
"UPDAT_PO"	SFC 27	SFC 27	// Update Outputs on I/O Module
"SET_TINT"	SFC 28	SFC 28	// Set Time-of-Day Interrupt
"CAN_TINT"	SFC 29	SFC 29	// Cancel Time-of-Day Interrupt
"ACT_TINT"	SFC 30	SFC 30	// Activate Time-of-Day Interrupt
"QRY_TINT"	SFC 31	SFC 31	// Query Time-of-Day Interrupt
"SRT_DINT"	SFC 32	SFC 32	// Start Time-Delay Interrupt
"CAN_DINT"	SFC 33	SFC 33	// Cancel Time-Delay Interrupt
"QRY_DINT"	SFC 34	SFC 34	// Query Time-Delay Interrupt
"MP_ALM"	SFC 35	SFC 35	// Trigger Multicomputing Interrupt
"MSK_FLT"	SFC 36	SFC 36	// Mask Synchronous Errors
"DMSK_FLT"	SFC 37	SFC 37	// Unmask Synchronous Errors
"READ_ERR"	SFC 38	SFC 38	// Read Error Registers
"DIS_IRT"	SFC 39	SFC 39	// Disable New Interrupts and Asynchronous Errors
"EN_IRT"	SFC 40	SFC 40	// Enable New Interrupts and Asynchronous Errors
"DIS_AIRT"	SFC 41	SFC 41	// Delay the Higher Priority Interrupts and Asynchronous Errors
"EN_AIRT"	SFC 42	SFC 42	// Enable Higher Priority Interrupts and Asynchronous Errors
"RE_TRIGR"	SFC 43	SFC 43	// Retrigger Cycle Time Monitoring
"REPL_VAL"	SFC 44	SFC 44	// Transfer Substitute Value to Accumulator 1
"STP"	SFC 46	SFC 46	// Change the CPU to STOP
"WAIT"	SFC 47	SFC 47	// Delay Execution of the User Program
"SNC_RTCB"	SFC 48	SFC 48	// Synchronize Slave Clocks
"LGC_GADR"	SFC 49	SFC 49	// Query the Module Slot Belonging to a Logical Address
"RD_LGADR"	SFC 50	SFC 50	// Read All Logical Addresses of a Module
"RDSYSST"	SFC 51	SFC 51	// Read a System Status List or Partial List
"WR_USMSG"	SFC 52	SFC 52	// Write a User-Defined Diagnostic Event to the Diagnostic Buffer
"RD_DPARM"	SFC 54	SFC 54	// Reading Predefined Parameters
"WR_PARM"	SFC 55	SFC 55	// Write Dynamic Parameters
"WR_DPARM"	SFC 56	SFC 56	// Write Default Parameters
"PARM_MOD"	SFC 57	SFC 57	// Assign Parameters to a Module
"WR_REC"	SFC 58	SFC 58	// Write Data Record
"RD_REC"	SFC 59	SFC 59	// Read a Data Record
"GD_SND"	SFC 60	SFC 60	// Send a GD Packet
"GD_RCV"	SFC 61	SFC 61	// Fetch a Received GD Packet
"CONTROL"	SFC 62	SFC 62	// Query the Status of a Connection Belonging to a Communication SFB Instance
"AB_CALL"	SFC 63	SFC 63	// Assembly Code Block (CPU 614)
"TIME_TCK"	SFC 64	SFC 64	// Read the System Time
"X_SEND"	SFC 65	SFC 65	// Send Data to a Communication Partner outside the Local S7 Station
"X_RCV"	SFC 66	SFC 66	// Receive Data from a Communication Partner outside the Local S7 Station
"X_GET"	SFC 67	SFC 67	// Read Data from a Communication Partner outside the Local S7 Station
"X_PUT"	SFC 68	SFC 68	// Write Data to a Communication Partner outside the Local S7 Station
"X_ABORT"	SFC 69	SFC 69	// Abort an Existing Connection to a  Partner outside the Local S7 Station
"I_GET"	SFC 72	SFC 72	// Read Data from a Communication Partner within the Local S7 Station
"I_PUT"	SFC 73	SFC 73	// Write Data to a Communication Partner within the Local S7 Station
"I_ABORT"	SFC 74	SFC 74	// Abort an Existing Connection to a Partner within the Local S7 Station
"DI_Vars"	VAT 1	
"DO_Vars"	VAT 2	
"AI_Vars"	VAT 3	
"AO_Vars"	VAT 4	
END_SYMBOL_TABLE
